PROGRAM Main
VAR
	// XRTM1
	// Motors
	{attribute 'TcLinkTo' := '.bLimitForwardEnable:=TIIB[EL7041-1000_XRTM1_Yup]^STM Status^Status^Digital input 1;
                              .bLimitBackwardEnable:=TIIB[EL7041-1000_XRTM1_Yup]^STM Status^Status^Digital input 2'}
	{attribute 'pytmc' := '
		pv: XRTMR1:HOMS:MMS:YUP
	'}
	M1 : DUT_MotionStage := (fVelocity:=200.0, nEnableMode:=ENUM_StageEnableMode.ALWAYS, bPowerSelf:=TRUE); // XRTM1 Yup
	fbMotionStage_m1 : FB_MotionStage;

	{attribute 'TcLinkTo' := '.bLimitForwardEnable:=TIIB[EL7041-1000_XRTM1_Ydwn]^STM Status^Status^Digital input 1;
                              .bLimitBackwardEnable:=TIIB[EL7041-1000_XRTM1_Ydwn]^STM Status^Status^Digital input 2'}
	{attribute 'pytmc' := '
		pv: XRTMR1:HOMS:MMS:YDWN
	'}
	M2 : DUT_MotionStage := (fVelocity:=200.0, nEnableMode:=ENUM_StageEnableMode.ALWAYS, bPowerSelf:=TRUE); // XRTM1 Ydwn
	fbMotionStage_m2 : FB_MotionStage;

	{attribute 'TcLinkTo' := '.bLimitForwardEnable:=TIIB[EL7041-1000_XRTM1_Xup]^STM Status^Status^Digital input 1;
                              .bLimitBackwardEnable:=TIIB[EL7041-1000_XRTM1_Xup]^STM Status^Status^Digital input 2'}
	{attribute 'pytmc' := '
		pv: XRTMR1:HOMS:MMS:XUP
	'}
	M3 : DUT_MotionStage := (fVelocity:=1000.0, nEnableMode:=ENUM_StageEnableMode.ALWAYS, bPowerSelf:=TRUE); // XRTM1 Xup
	fbMotionStage_m3 : FB_MotionStage;

	{attribute 'TcLinkTo' := '.bLimitForwardEnable:=TIIB[EL7041-1000_XRTM1_Xdwn]^STM Status^Status^Digital input 1;
                              .bLimitBackwardEnable:=TIIB[EL7041-1000_XRTM1_Xdwn]^STM Status^Status^Digital input 2'}
	{attribute 'pytmc' := '
		pv: XRTMR1:HOMS:MMS:XDWN
	'}
	M4 : DUT_MotionStage := (fVelocity:=1000.0, nEnableMode:=ENUM_StageEnableMode.ALWAYS, bPowerSelf:=TRUE); // XRTM1 Xdwn
	fbMotionStage_m4 : FB_MotionStage;

	{attribute 'TcLinkTo' := '.bLimitForwardEnable:=TIIB[EL7041-1000_XRTM1_PitchCoarse]^STM Status^Status^Digital input 1;
                              .bLimitBackwardEnable:=TIIB[EL7041-1000_XRTM1_PitchCoarse]^STM Status^Status^Digital input 2'}
	{attribute 'pytmc' := '
		pv: XRTMR1:HOMS:MMS:PITCH
	'}
	M5 : DUT_MotionStage := (fVelocity:=150.0); // XRTM1 Pitch Stepper

	{attribute 'TcLinkTo' := '.bLimitForwardEnable:=TIIB[EL7041-1000_XRTM1_Bender]^STM Status^Status^Digital input 1;
                              .bLimitBackwardEnable:=TIIB[EL7041-1000_XRTM1_Bender]^STM Status^Status^Digital input 2'}
	{attribute 'pytmc' := '
		pv: XRTMR1:HOMS:MMS:BENDER
	'}
	M6 : DUT_MotionStage := (fVelocity:=150.0, nEnableMode:=ENUM_StageEnableMode.ALWAYS, bPowerSelf:=TRUE); // XRTM1 Bender
	fbMotionStage_m6 : FB_MotionStage;

	{attribute 'TcLinkTo' := '.fbRunHOMS.bSTOEnable1:=TIIB[EL1004_XRTM1_STO]^Channel 1^Input;
                              .fbRunHOMS.bSTOEnable2:=TIIB[EL1004_XRTM1_STO]^Channel 2^Input;
	                          .fbRunHOMS.stYupEnc.Count:=TIIB[EL5042_XRTM1_Yupdwn]^FB Inputs Channel 1^Position;
	                          .fbRunHOMS.stYdwnEnc.Count:=TIIB[EL5042_XRTM1_Yupdwn]^FB Inputs Channel 2^Position;
	                          .fbRunHOMS.stXupEnc.Count:=TIIB[EL5042_XRTM1_Xupdwn]^FB Inputs Channel 1^Position;
	                          .fbRunHOMS.stXdwnEnc.Count:=TIIB[EL5042_XRTM1_Xupdwn]^FB Inputs Channel 2^Position'}
	{attribute 'pytmc' := '
		pv: XRTMR1:HOMS
	'}
	XRTM1 : DUT_HOMS;

	// Encoder Arrays/RMS Watch:
	{attribute 'pytmc' := '
		pv: XRTMR1:HOMS:ENC:Y
	'}
	fbYRMSErrorXRTM1 : FB_RMSWatch;
	fMaxYRMSErrorXRTM1 : LREAL;
	fMinYRMSErrorXRTM1 : LREAL;

	{attribute 'pytmc' := '
		pv: XRTMR1:HOMS:ENC:X
	'}
	fbXRMSErrorXRTM1 : FB_RMSWatch;
	fMaxXRMSErrorXRTM1 : LREAL;
	fMinXRMSErrorXRTM1 : LREAL;

	{attribute 'pytmc' := '
		pv: XRTMR1:HOMS:ENC:PITCH
	'}
	fbPitchRMSErrorXRTM1 : FB_RMSWatch;
	fMaxPitchRMSErrorXRTM1 : LREAL;
	fMinPitchRMSErrorXRTM1 : LREAL;

	{attribute 'pytmc' := '
		pv: XRTMR1:HOMS:ENC:BENDER
	'}
	fbBenderRMSErrorXRTM1 : FB_RMSWatch;
	fMaxBenderRMSErrorXRTM1 : LREAL;
	fMinBenderRMSErrorXRTM1 : LREAL;

	// Pitch Control
	fbXRTM1PitchControl : FB_PitchControl;
	bXRTM1PitchDone : BOOL;
	bXRTM1PitchBusy : BOOL;

	// Bender Control
	fbBenderXRTM1 : FB_Bender;

	// Raw Encoder Counts
	{attribute 'pytmc' := '
		pv: XRTMR1:HOMS:ENC:YUP:CNT
		field: EGU cnt
		io: i
	'}
	nEncCntYupXRTM1 : UDINT;
	{attribute 'pytmc' := '
		pv: XRTMR1:HOMS:ENC:YDWN:CNT
		field: EGU cnt
		io: i
	'}
	nEncCntYdwnXRTM1 : UDINT;
	{attribute 'pytmc' := '
		pv: XRTMR1:HOMS:ENC:XUP:CNT
		field: EGU cnt
		io: i
	'}
	nEncCntXupXRTM1 : UDINT;
	{attribute 'pytmc' := '
		pv: XRTMR1:HOMS:ENC:XDWN:CNT
		field: EGU cnt
		io: i
	'}
	nEncCntXdwnXRTM1 : UDINT;
	{attribute 'pytmc' := '
		pv: XRTMR1:HOMS:ENC:PITCH:CNT
		field: EGU cnt
		io: i
	'}
	nEncCntPitchXRTM1 : UDINT;

	// Encoder Reference Values
	{attribute 'pytmc' := '
		pv: XRTMR1:HOMS:ENC:YUP:REF
		field: EGU cnt
		io: i
	'}
	nEncRefYupXRTM1 : UDINT;
	{attribute 'pytmc' := '
		pv: XRTMR1:HOMS:ENC:YDWN:REF
		field: EGU cnt
		io: i
	'}
	nEncRefYdwnXRTM1 : UDINT;
	{attribute 'pytmc' := '
		pv: XRTMR1:HOMS:ENC:XUP:REF
		field: EGU cnt
		io: i
	'}
	nEncRefXupXRTM1 : UDINT;
	{attribute 'pytmc' := '
		pv: XRTMR1:HOMS:ENC:XDWN:REF
		field: EGU cnt
		io: i
	'}
	nEncRefXdwnXRTM1 : UDINT;
	{attribute 'pytmc' := '
		pv: XRTMR1:HOMS:ENC:PITCH:REF
		field: EGU cnt
		io: i
	'}
	nEncRefPitchXRTM1 : UDINT;
	mcReadParameterPitchXRTM1 : MC_ReadParameter;
	fEncRefPitchXRTM1_urad : LREAL; // Current Pitch encoder offset in urad
	
    //****** HOMS M2 and M3 **************************
	tpImAPLC : TP := (PT:=T#10S);
	ExpertMode	:	BOOL := FALSE;
	PitchManualMode: BOOL := FALSE;
	
	//Drive CoE Fb
	fbY1CoE	:	FB_ElmoGDCBellCoE;
	fbY2CoE	:	FB_ElmoGDCBellCoE;
	
	fbX1CoE	:	FB_ElmoGDCBellCoE;
	fbX2CoE	:	FB_ElmoGDCBellCoE;
	
	fbP1CoE	:	FB_ElmoGDCBellCoE;
	fbB1CoE	:	FB_ElmoGDCBellCoE;
	
	//Init params trigger
	rtInitParams	:	R_TRIG;
	
	//Test Parameters
	rStepSize: REAL;
	SettleTime: TON := (
	PT:=T#2s);
	TestUpperVoltage: REAL := 100;
	TestLowerVoltage: REAL := 10;
	xRunPiezoRepeatTest: BOOL;
	
	//Drive reference initializations
	fbInitDriveRef	:	FB_InitDriveRefs;
	//MPS Information
	fbMPS_States :  FB_MPS_STATES;
	M2_INRANGE  :   ARRAY[0..1] OF DINT := [24568920, 26568920];
	M2_OUTRANGE  :  ARRAY[0..1] OF DINT := [43568250, 50570250];
	//noConsequence	:	BOOL;
	
	mcBenderPower	:	MC_POWER;
	
	// HOMS M2
	XRTM2PitchControl	    :	FB_PitchControlOld;
	XRTM2Y_GantryControl	:	FB_Gantry;
	XRTM2X_GantryControl	:	FB_Gantry;
	
	fbM2Y1LS	:	FB_LimitSwitchState;
	fbM2Y2LS	:	FB_LimitSwitchState;
	fbM2X1LS	:	FB_LimitSwitchState;
	fbM2X2LS	:	FB_LimitSwitchState;
	fbM2P1LS	:	FB_PitchSoftLimits;	
	
    // HOMS M3
	XRTM3PitchControl	    :	FB_PitchControlOld;
	XRTM3Y_GantryControl	:	FB_Gantry;
	XRTM3X_GantryControl	:	FB_Gantry;
	
	fbM3Y1LS	:	FB_LimitSwitchState;
	fbM3Y2LS	:	FB_LimitSwitchState;
	fbM3X1LS	:	FB_LimitSwitchState;
	fbM3X2LS	:	FB_LimitSwitchState;
	fbM3P1LS	:	FB_PitchSoftLimits;	
	
	//************** **** *** ** *
	
	
	
	// PMPS arbiter interface
	fbArbiterIO : FB_SubSysToArbiter_IO;
	
	// Common
	fEncLeverArm_mm : LREAL := 513.0;
	// Logging
	fbLogHandler : FB_LogHandler;

END_VAR

// XRTM1
XRTM1.fbRunHOMS(stYup:=M1,
               stYdwn:=M2,
               stXup:=M3,
               stXdwn:=M4,
               stPitch:=M5,
	           nYupEncRef:=GVL_XRTM1_Constants.nYUP_ENC_REF,
               nYdwnEncRef:=GVL_XRTM1_Constants.nYDWN_ENC_REF,
               nXupEncRef:=GVL_XRTM1_Constants.nXUP_ENC_REF,
               nXdwnEncRef:=GVL_XRTM1_Constants.nXDWN_ENC_REF,
			   bExecuteCoupleY:=XRTM1.bExecuteCoupleY,
               bExecuteCoupleX:=XRTM1.bExecuteCoupleX,
			   bExecuteDecoupleY:=XRTM1.bExecuteDecoupleY,
               bExecuteDecoupleX:=XRTM1.bExecuteDecoupleX,
               bGantryAlreadyCoupledY=>XRTM1.bGantryAlreadyCoupledY,
               bGantryAlreadyCoupledX=>XRTM1.bGantryAlreadyCoupledX,
               nCurrGantryY=>XRTM1.nCurrGantryY,
               nCurrGantryX=>XRTM1.nCurrGantryX);
fbBenderXRTM1(stBender:=M6,
	         bSTOEnable1:=XRTM1.fbRunHOMS.bSTOEnable1,
		     bSTOEnable2:=XRTM1.fbRunHOMS.bSTOEnable2);
// No slave motion through Epics
M2.bExecute := FALSE; // XRTM1-Ydwn
M4.bExecute := FALSE; // XRTM1-Xdwn

// Convert nCurrGantry to um (smaller number) to read out in epics
XRTM1.fCurrGantryY_um := LINT_TO_REAL(XRTM1.nCurrGantryY) / 1000.0;
XRTM1.fCurrGantryX_um := LINT_TO_REAL(XRTM1.nCurrGantryX) / 1000.0;

// FB_MotionStage's for non-piezo axes
fbMotionStage_m1(stMotionStage:=M1);
fbMotionStage_m2(stMotionStage:=M2);
fbMotionStage_m3(stMotionStage:=M3);
fbMotionStage_m4(stMotionStage:=M4);
fbMotionStage_m6(stMotionStage:=M6);

// Calculate Pitch RMS Error:
fbYRMSErrorXRTM1(stMotionStage:=M1,
	            fMaxRMSError=>fMaxYRMSErrorXRTM1,
				fMinRMSError=>fMinYRMSErrorXRTM1);

fbXRMSErrorXRTM1(stMotionStage:=M3,
	            fMaxRMSError=>fMaxXRMSErrorXRTM1,
				fMinRMSError=>fMinXRMSErrorXRTM1);

fbPitchRMSErrorXRTM1(stMotionStage:=M5,
	                fMaxRMSError=>fMaxPitchRMSErrorXRTM1,
					fMinRMSError=>fMinPitchRMSErrorXRTM1);

fbBenderRMSErrorXRTM1(stMotionStage:=M6,
	                 fMaxRMSError=>fMaxBenderRMSErrorXRTM1,
					 fMinRMSError=>fMinBenderRMSErrorXRTM1);
// Pitch Control
fbXRTM1PitchControl(Pitch:=GVL_XRTM1.XRTM1_Pitch,
				   Stepper:=M5,
				   lrCurrentSetpoint:=M5.fPosition,
                   q_bDone=>bXRTM1PitchDone,
                   q_bBusy=>bXRTM1PitchBusy);
// When STO hit, need to reset SP
IF NOT M5.bHardwareEnable THEN
	M5.fPosition := M5.stAxisStatus.fActPosition;
END_IF

// Raw Encoder Counts For Epics
nEncCntYupXRTM1 := ULINT_TO_UDINT(XRTM1.fbRunHOMS.stYupEnc.Count);
nEncCntYdwnXRTM1 := ULINT_TO_UDINT(XRTM1.fbRunHOMS.stYdwnEnc.Count);
nEncCntXupXRTM1 := ULINT_TO_UDINT(XRTM1.fbRunHOMS.stXupEnc.Count);
nEncCntXdwnXRTM1 := ULINT_TO_UDINT(XRTM1.fbRunHOMS.stXdwnEnc.Count);
nEncCntPitchXRTM1 := LINT_TO_UDINT(GVL_XRTM1.XRTM1_Pitch.diEncCnt);

// Encoder Reference Values For Epics
nEncRefYupXRTM1 := ULINT_TO_UDINT(GVL_XRTM1_Constants.nYUP_ENC_REF);
nEncRefYdwnXRTM1 := ULINT_TO_UDINT(GVL_XRTM1_Constants.nYDWN_ENC_REF);
nEncRefXupXRTM1 := ULINT_TO_UDINT(GVL_XRTM1_Constants.nXUP_ENC_REF);
nEncRefXdwnXRTM1 := ULINT_TO_UDINT(GVL_XRTM1_Constants.nXDWN_ENC_REF);
mcReadParameterPitchXRTM1(Axis:=M5.Axis,
	                     Enable:=TRUE,
				         ParameterNumber:=MC_AxisParameter.AxisEncoderOffset,
				         ReadMode:=READMODE_CYCLIC,
				         Value=>fEncRefPitchXRTM1_urad);

nEncRefPitchXRTM1 := LREAL_TO_UDINT(ABS(fEncRefPitchXRTM1_urad) * fEncLeverArm_mm);

// HOMS ************************ ***** **** *** ** *
p_ModbusRx_OutputCoils();
p_ModbusRx_PLCMemory();

//InitParams
////////////////////
rtInitParams(CLK:=gFirstPass);
IF rtInitParams.Q THEN
	Init_XRTM2();
	Init_XRTM3();
	gFirstPass := FALSE;
END_IF

//System Error Handling
/////////////////////////////////////
//SystemErrorSummary(); //Check this action for a summary of all system faults
					  
//SystemError();

//Driver Parameter Verification
/////////////////////////////////////

//Gantry Interlock Logic
/////////////////////////////////////
	//SimGantry.VAxis.i_xMotorInterlock := TRUE;
	//SimGantry.PAxis.i_xMotorInterlock := TRUE;
	//SimGantry.SAxis.i_xMotorInterlock := TRUE;
	
LimitSwitchIO();

// Pitch control
/////////////////////////////////////
XRTM2PitchControl(Pitch:=HOMS2_Pitch, DirectPiezoMode:=(ExpertMode AND PitchManualMode), q_xDone=>HOMS2_Pitch.Axis.bDone, q_xBusy => HOMS2_Pitch.Axis.bBusy);
XRTM3PitchControl(Pitch:=HOMS3_Pitch, DirectPiezoMode:=(ExpertMode AND PitchManualMode), q_xDone=>HOMS3_Pitch.Axis.bDone, q_xBusy => HOMS3_Pitch.Axis.bBusy);
//Y motion
/////////////////////////////////////
HOMS3_YGantry.PAxis.stAxis.ReadStatus();
HOMS3_YGantry.SAxis.stAxis.ReadStatus();
HOMS3_YGantry.PAxis.stStatus.rActPosition := LREAL_TO_REAL(HOMS3_YGantry.PAxis.stAxis.NcToPlc.ActPos);
HOMS3_YGantry.SAxis.stStatus.rActPosition := LREAL_TO_REAL(HOMS3_YGantry.SAxis.stAxis.NcToPlc.ActPos);

//X Motion
/////////////////////////////////////
XRTM2X_GantryControl(Gantry:=HOMS2_XGantry);
XRTM3X_GantryControl(Gantry:=HOMS3_XGantry);

//Communicate state to MPS
////////////////////////////////
fbMPS_States(GANTRY:=HOMS2_XGantry,
			 OUT_LS:=NOT HOMS2_XGantry.PAxis.xHiLS OR NOT HOMS2_XGantry.SAxis.xLoLS,
			 IN_RANGE:=M2_INRANGE,
			 OUT_RANGE:=M2_OUTRANGE);
			 
bXRT_M2_IN  := fbMPS_States.IN;
bXRT_M2_OUT := fbMPS_States.OUT;
//EPICS Tx Update
////////////////////
p_ModbusTx_InputCoils();
//p_ModbusTx_OutputCoils();
p_ModbusTx_InputReg();
p_ModbusTx_PLCMemory();

// **************************** ***** **** *** ** * HOMS


P_CoatingProtections();

// Logging
fbLogHandler();

// PMPS
GVL_PMPS.g_fbArbiter1.AddRequest(16#5, PMPS_GVL.cstFullBeam);
fbArbiterIO(Arbiter := GVL_PMPS.g_fbArbiter1, fbFFHWO := GVL_PMPS.g_FastFaultOutput1);
GVL_PMPS.g_FastFaultOutput1.Execute(i_xVeto:=);
GVL_PMPS.g_FastFaultOutput2.Execute(i_xVeto:=);

ACTION Init_XRTM2:
//FEE-M2
///////////////////////////


//Initialize ELMO Drive references
fbInitDriveRef(stCoE:=HOMS2_XGantry.PAxis.stCoE);
fbInitDriveRef(stCoE:=HOMS2_XGantry.SAxis.stCoE);
fbInitDriveRef(stCoE:=HOMS2_YGantry.PAxis.stCoE);
fbInitDriveRef(stCoE:=HOMS2_YGantry.SAxis.stCoE);
fbInitDriveRef(stCoE:=HOMS2_Pitch.Stepper.stCoE);

//Initialze Drive Speeds and Accelerations
//////////////////////////////////////////
HOMS2_XGantry.PAxis.fAcceleration := 1.0;
HOMS2_XGantry.SAxis.fAcceleration := 1.0;
HOMS2_YGantry.PAxis.fAcceleration := 1.0;
HOMS2_YGantry.SAxis.fAcceleration := 1.0;

HOMS2_XGantry.PAxis.fDeceleration := 1.0;
HOMS2_XGantry.SAxis.fDeceleration := 1.0;
HOMS2_YGantry.PAxis.fDeceleration := 1.0;
HOMS2_YGantry.SAxis.fDeceleration := 1.0;

HOMS2_XGantry.PAxis.fVelocity := 0.1;
HOMS2_XGantry.SAxis.fVelocity := 0.1;
HOMS2_YGantry.PAxis.fVelocity := 0.1;
HOMS2_YGantry.SAxis.fVelocity := 0.1;

HOMS2_Pitch.Stepper.fAcceleration := 39;
HOMS2_Pitch.Stepper.fDeceleration := 39;
HOMS2_Pitch.Stepper.fVelocity     := 100;

//Initialize Piezo Driver
/////////////////////////////////////
HOMS2_Pitch.Piezo.stPIParams.fKp := 0.001;
HOMS2_Pitch.Piezo.stPIParams.tTn := T#500MS;
HOMS2_Pitch.Piezo.stPIParams.fOutMaxLimit := 1;
HOMS2_Pitch.Piezo.stPIParams.fOutMinLimit := -1;
END_ACTION

ACTION Init_XRTM3:
//FEE-M3
///////////////////////////


//Initialize ELMO Drive references
fbInitDriveRef(stCoE:=HOMS3_XGantry.PAxis.stCoE);
fbInitDriveRef(stCoE:=HOMS3_XGantry.SAxis.stCoE);
fbInitDriveRef(stCoE:=HOMS3_YGantry.PAxis.stCoE);
fbInitDriveRef(stCoE:=HOMS3_YGantry.SAxis.stCoE);
fbInitDriveRef(stCoE:=HOMS3_Pitch.Stepper.stCoE);

//Initialze Drive Speeds and Accelerations
//////////////////////////////////////////
HOMS3_XGantry.PAxis.fAcceleration := 1.0;
HOMS3_XGantry.SAxis.fAcceleration := 1.0;
HOMS3_YGantry.PAxis.fAcceleration := 1.0;
HOMS3_YGantry.SAxis.fAcceleration := 1.0;

HOMS3_XGantry.PAxis.fDeceleration := 1.0;
HOMS3_XGantry.SAxis.fDeceleration := 1.0;
HOMS3_YGantry.PAxis.fDeceleration := 1.0;
HOMS3_YGantry.SAxis.fDeceleration := 1.0;

HOMS3_XGantry.PAxis.fVelocity := 0.1;
HOMS3_XGantry.SAxis.fVelocity := 0.1;
HOMS3_YGantry.PAxis.fVelocity := 0.1;
HOMS3_YGantry.SAxis.fVelocity := 0.1;

HOMS3_Pitch.Stepper.fAcceleration := 39;
HOMS3_Pitch.Stepper.fDeceleration := 39;
HOMS3_Pitch.Stepper.fVelocity     := 100;

//Initialize Piezo Driver
/////////////////////////////////////
HOMS3_Pitch.Piezo.stPIParams.fKp := 0.001;
HOMS3_Pitch.Piezo.stPIParams.tTn := T#500MS;
HOMS3_Pitch.Piezo.stPIParams.fOutMaxLimit := 1;
HOMS3_Pitch.Piezo.stPIParams.fOutMinLimit := -1;
END_ACTION

ACTION LimitSwitchIO:
//XRT M2
//////////////////////////
fbM2Y1LS(diInputs:=HOMS2_YGantry.PAxis.diInputs, 
xHiLS=>HOMS2_YGantry.PAxis.xHiLS,
xLoLS=>HOMS2_YGantry.PAxis.xLoLS,
STO => gM2STO);

fbM2Y2LS(diInputs:=HOMS2_YGantry.SAxis.diInputs, 
xHiLS=>HOMS2_YGantry.SAxis.xHiLS,
xLoLS=>HOMS2_YGantry.SAxis.xLoLS);

fbM2X1LS(diInputs:=HOMS2_XGantry.PAxis.diInputs, 
xHiLS=>HOMS2_XGantry.PAxis.xHiLS,
xLoLS=>HOMS2_XGantry.PAxis.xLoLS);

fbM2X2LS(diInputs:=HOMS2_XGantry.SAxis.diInputs, 
xHiLS=>HOMS2_XGantry.SAxis.xHiLS,
xLoLS=>HOMS2_XGantry.SAxis.xLoLS);

fbM2P1LS(Pitch:=HOMS2_Pitch,
xHiLS=>HOMS2_Pitch.Stepper.xHiLS,
xLoLS=>HOMS2_Pitch.Stepper.xLoLS);

//XRT M3
//////////////////////////
fbM3Y1LS(diInputs:=HOMS3_YGantry.PAxis.diInputs, 
xHiLS=>HOMS3_YGantry.PAxis.xHiLS,
xLoLS=>HOMS3_YGantry.PAxis.xLoLS,
STO => gM3STO);

fbM3Y2LS(diInputs:=HOMS3_YGantry.SAxis.diInputs, 
xHiLS=>HOMS3_YGantry.SAxis.xHiLS,
xLoLS=>HOMS3_YGantry.SAxis.xLoLS);

fbM3X1LS(diInputs:=HOMS3_XGantry.PAxis.diInputs, 
xHiLS=>HOMS3_XGantry.PAxis.xHiLS,
xLoLS=>HOMS3_XGantry.PAxis.xLoLS);
(*
fbM3X2LS(diInputs:=HOMS3_XGantry.PAxis.diInputs,  //Paxis is here on purpose <HACK>
xHiLS=>HOMS3_XGantry.SAxis.xHiLS,
xLoLS=>HOMS3_XGantry.SAxis.xLoLS);
*)
fbM3X2LS(diInputs:=HOMS3_XGantry.SAxis.diInputs,  // Switching to SAxis works as expected, reason for <HACK> unclear
xHiLS=>HOMS3_XGantry.SAxis.xHiLS,
xLoLS=>HOMS3_XGantry.SAxis.xLoLS);

fbM3P1LS(Pitch:=HOMS3_Pitch,
xHiLS=>HOMS3_Pitch.Stepper.xHiLS,
xLoLS=>HOMS3_Pitch.Stepper.xLoLS);
END_ACTION

END_PROGRAM

(* stored: Version 1.1.0.1, ProductVersion 3.1.4024.6
   POU Main: Id {371c560d-bfd7-44d3-85a8-59ca1fa1938a}, SpecialFunc None
   Action Init_XRTM2: Id {5f4f0886-bfe6-466e-ab0f-beab0308d09d}
   Action Init_XRTM3: Id {4cd8bf74-eac1-478e-83ee-065628004dc5}
   Action LimitSwitchIO: Id {f9e468fa-ee02-4f8a-956e-139b70621257} *)
